(* IEC 61131-3 sources: programs/VI-54/VI-54_20171205/VI-54_20171205/Stations/Screen/LseClass170718/Class/inpSetPositions, 1 file *)

(* ---- inpSetPositions.st ---- *)
(*!
<Class
	Name               = "inpSetPositions"
	Revision           = "0.0"
	RealtimeTask       = "false"
	CyclicTask         = "false"
	BackgroundTask     = "false"
	Sigmatek           = "false"
	OSInterface        = "false"
	HighPriority       = "false"
	Automatic          = "false"
	UpdateMode         = "Prescan"
	SharedCommandTable = "true"
	Objectsize         = "(900,120)">
	<Channels>
		<Server Name="ButtonChoice" Visualized="true" Initialize="false" WriteProtected="false" Retentive="false"/>
		<Server Name="PosError" Visualized="true" Initialize="false" WriteProtected="true" Retentive="false"/>
		<Server Name="Rpos" Visualized="true" Initialize="false" WriteProtected="false" Retentive="false"/>
		<Server Name="SetNbr" Visualized="true" Initialize="false" WriteProtected="false" Retentive="false"/>
		<Server Name="Xpos" Visualized="true" Initialize="false" WriteProtected="false" Retentive="false"/>
		<Server Name="Ypos" Visualized="true" Initialize="false" WriteProtected="false" Retentive="false"/>
		<Server Name="Zpos" Visualized="true" Initialize="false" WriteProtected="false" Retentive="false"/>
		<Client Name="Model" Required="true" Internal="false"/>
		<Client Name="PositionChain" Required="false" Internal="false"/>
		<Client Name="PositionCheck" Required="true" Internal="false"/>
		<Client Name="TerminalControl" Required="true" Internal="false"/>
	</Channels>
	<Network Name="inpSetPositions">
		<!-- List of Components in this network -->
		<Components>
			<Object
				Name       = "_base"
				Class      = "ReceptBase"
				Position   = "(218,120)"
				Visualized = "false">
				<Channels>
					<Server Name="Refresh"/>
					<Server Name="Size"/>
					<Client Name="Data"/>
				</Channels>
			</Object>
		</Components>
		<Comments>
		</Comments>
		<!-- List of Connections in this network -->
		<Connections>
			<Connection Source="_base.Data" Destination="this.Data" Vertices="(218,210),(38,210),"/>
			<Connection Source="this.Refresh" Destination="_base.Refresh" Vertices="(690,210),(518,210),"/>
		</Connections>
		<!-- Headerfiles -->
		<Options>
		</Options>
	</Network>
</Class>
*)
#pragma using ReceptBase

inpSetPositions : CLASS
: ReceptBase
  //Servers:
	ButtonChoice 	: SvrCh_DINT;
	SetNbr 	: SvrCh_DINT;
	Xpos 	: SvrCh_DINT;
	Zpos 	: SvrCh_DINT;
	Rpos 	: SvrCh_DINT;
	Ypos 	: SvrCh_DINT;
	PosError 	: SvrCh_DINT;
  //Clients:
	Model 	: CltChCmd_ModelD4V2;
	TerminalControl 	: CltChCmd_TerminalControl;
	PositionCheck 	: CltChCmd_GetLimits;
	PositionChain 	: CltChCmd_Position;
  //Variables:
		ButtonChoiceTmr 	: UDINT;
		GiveCommandOnes 	: DINT;
  //Functions:

	FUNCTION VIRTUAL GLOBAL Init;

	FUNCTION VIRTUAL GLOBAL RefreshPara;

	FUNCTION GLOBAL ChoiceCheck;

	FUNCTION GLOBAL SetPosNbr
		VAR_INPUT
			Nbr 	: DINT;
		END_VAR;

	FUNCTION GLOBAL CheckWindow
		VAR_INPUT
			WindowNbr 	: DINT;
		END_VAR
		VAR_OUTPUT
			State 	: DINT;
		END_VAR;

	FUNCTION CheckPositions
		VAR_INPUT
			Positions 	: _LMCPROF_POS;
		END_VAR
		VAR_OUTPUT
			Retcode 	: BOOL;
		END_VAR;
  //Tables:
	FUNCTION @STD
		VAR_OUTPUT
			ret_code	: CONFSTATES;
		END_VAR;
	FUNCTION GLOBAL TAB @CT_;
END_CLASS;

#pragma usingLtd GetLimits
#pragma usingLtd ModelD4V2
#pragma usingLtd Position
#pragma usingLtd TerminalControl

FUNCTION VIRTUAL GLOBAL inpSetPositions::Init

  PositionChain.PosNbr(inpNbr:= 1);

  if _FirstScan = 1 then
    ReceptPtr$^Usint := Data.GetDataPtr();
    PositionChain.SetRecipePtr(Ptr:= ReceptPtr);
  end_if;

END_FUNCTION

FUNCTION VIRTUAL GLOBAL inpSetPositions::RefreshPara

  // Refresh the parameters
  Xpos    := ReceptPtr^.RobotPositions[SetNbr].Xpos;
  Ypos    := ReceptPtr^.RobotPositions[SetNbr].Ypos;
  Zpos    := ReceptPtr^.RobotPositions[SetNbr].Zpos;
  Rpos    := ReceptPtr^.RobotPositions[SetNbr].Rpos;

END_FUNCTION

FUNCTION GLOBAL inpSetPositions::ChoiceCheck
  VAR
  	positions : _LMCPROF_POS;
  END_VAR

  if ButtonChoice <> 0 then
    if (ops.tAbsolute - ButtonChoiceTmr) >= 500 then
      if ButtonChoice >= 2 then // dubble click
        if CheckWindow(WindowNbr:= 201) = True then
          SetNbr := -1;
          ButtonChoice := 0;
        end_if;
      else // set position
        Model.GetRobotPosition(Mode:=_LMCRobotBase::_POSITION_MODE::_SETPOS_APPUNITS, IncludeTool:=0, CoordSystem:=0, pPositions:=#positions);
        if SetNbr <> -1 then
          // Check position and set positions
          if CheckPositions(Positions:= positions) = True then
            PosError := 0;
            ReceptPtr^.RobotPositions[SetNbr].Xpos := Positions.Pos1;
            ReceptPtr^.RobotPositions[SetNbr].Ypos := Positions.Pos2;
            ReceptPtr^.RobotPositions[SetNbr].Zpos := Positions.Pos3;
            ReceptPtr^.RobotPositions[SetNbr].Rpos := Positions.Pos4;

            // Set to chain
            PositionChain.PosData(inpData:= ReceptPtr^.RobotPositions[SetNbr], inpNbr:= SetNbr);
            RefreshPara();
          else // give window position error
            TerminalControl.SelectWindowNbr(Nbr:= 202);
          end_if;
        end_if;
        SetNbr := -1;
        ButtonChoice := 0;
      end_if;
    end_if;
  else
    ButtonChoiceTmr := ops.tAbsolute;
  end_if;

END_FUNCTION

FUNCTION GLOBAL inpSetPositions::SetPosNbr
	VAR_INPUT
		Nbr 	: DINT;
	END_VAR

  SetNbr := Nbr;

END_FUNCTION

FUNCTION GLOBAL inpSetPositions::CheckWindow
	VAR_INPUT
		WindowNbr 	: DINT;
	END_VAR
	VAR_OUTPUT
		State 	: DINT;
	END_VAR

  State := FALSE;

  if TerminalControl.ActWindowNbr = WindowNbr then
    GiveCommandOnes := 0;
    State := TRUE;
  else
    if GiveCommandOnes <> 1 then
      TerminalControl.SelectWindowNbr(Nbr:= WindowNbr);
      GiveCommandOnes := 1;
    end_if;
  end_if;

END_FUNCTION

FUNCTION inpSetPositions::CheckPositions
	VAR_INPUT
		Positions 	: _LMCPROF_POS;
	END_VAR
	VAR_OUTPUT
		Retcode 	: BOOL;
	END_VAR

  Retcode := False;

  if (Positions.Pos1 < PositionCheck.SwMaxXas_units) & (Positions.Pos1 > PositionCheck.SwMinXas_units) then
    if (Positions.Pos2 < PositionCheck.SwMaxYas_units) & (Positions.Pos2 > PositionCheck.SwMinYas_units) then
      if (Positions.Pos3 < PositionCheck.SwMaxZas_units) & (Positions.Pos3 > PositionCheck.SwMinZas_units) then
        if (Positions.Pos4 < PositionCheck.SwMaxRas_units) & (Positions.Pos4 > PositionCheck.SwMinRas_units) then
          Retcode := True;
        else
          PosError := 4;
        end_if;
      else
        PosError := 3;
      end_if;
    else
      PosError := 2;
    end_if;
  else
    PosError := 1;
  end_if;

END_FUNCTION
